(* PLC project Tc2_Standard.WCONCAT Demo, tc3-libraries-kb TwinCAT 3.1 *)
(* stored: creationDateTime 2026-05-10T08:00:00, modificationDateTime 2026-05-10T08:00:00 *)

PROGRAM P_Demo_WCONCAT
  VAR
    sResult : WSTRING;  (* WCONCAT 的返回值（监视） *)
    bRun : BOOL;  (* 触发一次 WCONCAT 调用 *)
  END_VAR

            // ============================================================
// Tc2_Standard.WCONCAT 演示程序（FUNCTION）
// ============================================================
// 场景：对 WSTRING 执行 CONCAT 操作
// 验证步骤：
//   1. 编译并登录目标
//   2. 强制 bRun := TRUE 一个周期
//   3. 观察 sResult = "SUSWILLI"
//   4. bRun 自动复位
// ============================================================

IF bRun THEN
    sResult := WCONCAT("SUS","WILLI");
    bRun := FALSE;
END_IF;

          
END_PROGRAM
